FUNCTION FU_Scale_IO : BOOL
VAR_INPUT
END_VAR
VAR
	fbScale : FB_12bIntToReal;
END_VAR

fbScale(nInput:=INPUT.nXc, fMin:=0, fMax:=0.5, fOutput => ScaledInputs.fXc);
fbScale(nInput:=INPUT.nPS, fMin:=0, fMax:=400, fOutput => ScaledInputs.fPS);
fbScale(nInput:=INPUT.nPR, fMin:=0, fMax:=40, fOutput => ScaledInputs.fPR);
fbScale(nInput:=INPUT.nPC_A, fMin:=0, fMax:=400, fOutput => ScaledInputs.fPC_A);
fbScale(nInput:=INPUT.nPC_B, fMin:=0, fMax:=400, fOutput => ScaledInputs.fPC_B);
fbScale(nInput:=INPUT.nPW_A, fMin:=0, fMax:=400, fOutput => ScaledInputs.fPW_A);
fbScale(nInput:=INPUT.nPW_A1, fMin:=0, fMax:=400, fOutput => ScaledInputs.fPW_A1);
fbScale(nInput:=INPUT.nPW_B, fMin:=0, fMax:=400, fOutput => ScaledInputs.fPW_B);
fbScale(nInput:=INPUT.nPW_B1, fMin:=0, fMax:=400, fOutput => ScaledInputs.fPW_B1);
fbScale(nInput:=INPUT.nPW_D, fMin:=0, fMax:=40, fOutput => ScaledInputs.fPW_D);
fbScale(nInput:=INPUT.nQW, fMin:=-150, fMax:=150, fOutput => ScaledInputs.fQw);

END_FUNCTION

(* stored: Version 1.1.0.1, ProductVersion 3.1.4024.12
   POU FU_Scale_IO: Id {bb59701a-6b46-4e16-b928-e79921db74f8}, SpecialFunc None *)
